// TIA Portal V18 export
VAR_GLOBAL   // PLC tag table "10_CT-4"
   "iCT-4p" AT %I8.1 : Bool;
   "iCT-4" AT %I8.2 : Bool;
   "oCT-4p" AT %Q0.6 : Bool;
   "oCT-4" AT %Q0.7 : Bool;
END_VAR
